// TwinCAT 3 PLC project PLC1
// ProgramVersion: 3.1.4023.0
// libraries:
//   Tc2_Standard, * (Beckhoff Automation GmbH)
//   Tc2_System, * (Beckhoff Automation GmbH)
//   Tc3_Module, * (Beckhoff Automation GmbH)
// project tree:
//   / PlcTask.TcTTO
//   POUs/ MAIN.TcPOU, LadderExample.TcPOU
// real-time tasks:
//   TASK PlcTask: cycle T#10ms, priority 20, ADS port 350

CONFIGURATION PLC1
    RESOURCE PLC ON TwinCAT3
        TASK PlcTask(INTERVAL := T#10ms, PRIORITY := 20);
        PROGRAM MAIN WITH PlcTask : MAIN;
    END_RESOURCE
END_CONFIGURATION

// ---- POUs/MAIN.TcPOU
PROGRAM MAIN
VAR
	nCounter : INT := 0;
	nCounter3 : INT := 0;
END_VAR

nCounter:= nCounter + 1;
nCounter3:= nCounter + 10;

END_PROGRAM

// ---- POUs/LadderExample.TcPOU
PROGRAM LadderExample
VAR
	input: BOOL;
	output: BOOL;
END_VAR

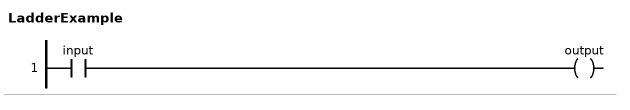
// NETWORK 1
output := input;

END_PROGRAM
